SUBAPPLICATION Uebung_152 (* Impulszähler & PI Regler *)
  (* Standard: 61499-2; Description: Copyright (c) 2023 Meisterschulen am Ostbahnhof This program and the accompanying materials are made available under the terms of the Eclipse Public License 2.0 which is available at https://www.eclipse.org/legal/epl-2.0/ SPDX-License-Identifier: EPL-2.0 *)
  (* Version 1.0, 2023-10-23, Franz Höpfinger, Meisterschulen am Ostbahnhof, initial API and implementation and/or initial documentation *)
  PACKAGE Uebungen;
  IMPORT logiBUS::io::DI::logiBUS_DI::Input_I1;
  IMPORT logiBUS::io::DI::logiBUS_DI::Input_I2;
  IMPORT logiBUS::io::DI::logiBUS_DI::Input_I3;
  IMPORT logiBUS::io::DI::logiBUS_DI_Events::BUTTON_SINGLE_CLICK;
  IMPORT logiBUS::io::DQ::logiBUS_DO::Output_Q1;
  IMPORT logiBUS::io::PI::logiBUS_PI::PulseInput_I8;
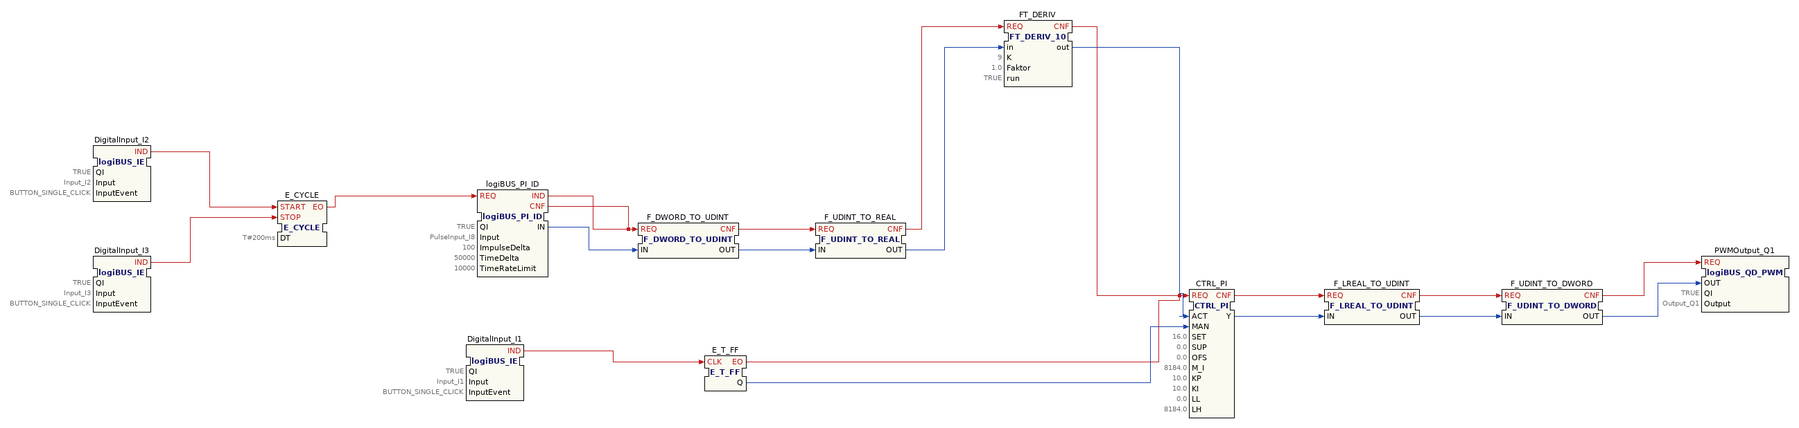
  FBS
    logiBUS_PI_ID : logiBUS::io::PI::logiBUS_PI_ID(QI := TRUE, Input := PulseInput_I8, ImpulseDelta := 100, TimeDelta := 50000, TimeRateLimit := 10000);
    FT_DERIV : OSCAT::Basic::POUs::Engineering::Control::FT_DERIV_10(K := 9, Faktor := 1.0, run := TRUE);
    F_DWORD_TO_UDINT : iec61131::conversion::F_DWORD_TO_UDINT;
    F_UDINT_TO_REAL : iec61131::conversion::F_UDINT_TO_REAL;
    PWMOutput_Q1 : logiBUS::io::DQ::logiBUS_QD_PWM(QI := TRUE, Output := Output_Q1);
    CTRL_PI : OSCAT::Basic::POUs::Engineering::Control::CTRL_PI(SET := 16.0, SUP := 0.0, OFS := 0.0, M_I := 8184.0, KP := 10.0, KI := 10.0, LL := 0.0, LH := 8184.0);
    DigitalInput_I1 : logiBUS::io::DI::logiBUS_IE(QI := TRUE, Input := Input_I1, InputEvent := BUTTON_SINGLE_CLICK);
    E_T_FF : iec61499::events::E_T_FF;
    F_LREAL_TO_UDINT : iec61131::conversion::F_LREAL_TO_UDINT;
    F_UDINT_TO_DWORD : iec61131::conversion::F_UDINT_TO_DWORD;
    E_CYCLE : iec61499::events::E_CYCLE(DT := T#200ms);
    DigitalInput_I2 : logiBUS::io::DI::logiBUS_IE(QI := TRUE, Input := Input_I2, InputEvent := BUTTON_SINGLE_CLICK);
    DigitalInput_I3 : logiBUS::io::DI::logiBUS_IE(QI := TRUE, Input := Input_I3, InputEvent := BUTTON_SINGLE_CLICK);
  END_FBS
  EVENT_CONNECTIONS
    logiBUS_PI_ID.IND TO F_DWORD_TO_UDINT.REQ;
    F_DWORD_TO_UDINT.CNF TO F_UDINT_TO_REAL.REQ;
    F_UDINT_TO_REAL.CNF TO FT_DERIV.REQ;
    FT_DERIV.CNF TO CTRL_PI.REQ;
    DigitalInput_I1.IND TO E_T_FF.CLK;
    E_T_FF.EO TO CTRL_PI.REQ;
    CTRL_PI.CNF TO F_LREAL_TO_UDINT.REQ;
    F_LREAL_TO_UDINT.CNF TO F_UDINT_TO_DWORD.REQ;
    F_UDINT_TO_DWORD.CNF TO PWMOutput_Q1.REQ;
    DigitalInput_I2.IND TO E_CYCLE.START;
    DigitalInput_I3.IND TO E_CYCLE.STOP;
    logiBUS_PI_ID.CNF TO F_DWORD_TO_UDINT.REQ;
    E_CYCLE.EO TO logiBUS_PI_ID.REQ;
  END_CONNECTIONS
  DATA_CONNECTIONS
    logiBUS_PI_ID.IN TO F_DWORD_TO_UDINT.IN;
    F_DWORD_TO_UDINT.OUT TO F_UDINT_TO_REAL.IN;
    F_UDINT_TO_REAL.OUT TO FT_DERIV.in;
    FT_DERIV.out TO CTRL_PI.ACT;
    E_T_FF.Q TO CTRL_PI.MAN;
    CTRL_PI.Y TO F_LREAL_TO_UDINT.IN;
    F_LREAL_TO_UDINT.OUT TO F_UDINT_TO_DWORD.IN;
    F_UDINT_TO_DWORD.OUT TO PWMOutput_Q1.OUT;
  END_CONNECTIONS
END_SUBAPPLICATION
